// TIA Portal V18 export
ORGANIZATION_BLOCK "OLDRestart"   // OB124, LAD, ProgramCycle
TITLE = "Main Program Sweep (Cycle)"
{ S7_Optimized_Access := 'TRUE' }
VERSION : 0.1
// stored: AutoNumber true, IsIECCheckEnabled false, SetENOAutomatically false
   VAR_INPUT
      Initial_Call : Bool;   // Initial call of this OB
      Remanence : Bool;   // =True, if remanent data are available
   END_VAR
BEGIN

REGION Network 1: RESTART CMMO Z2
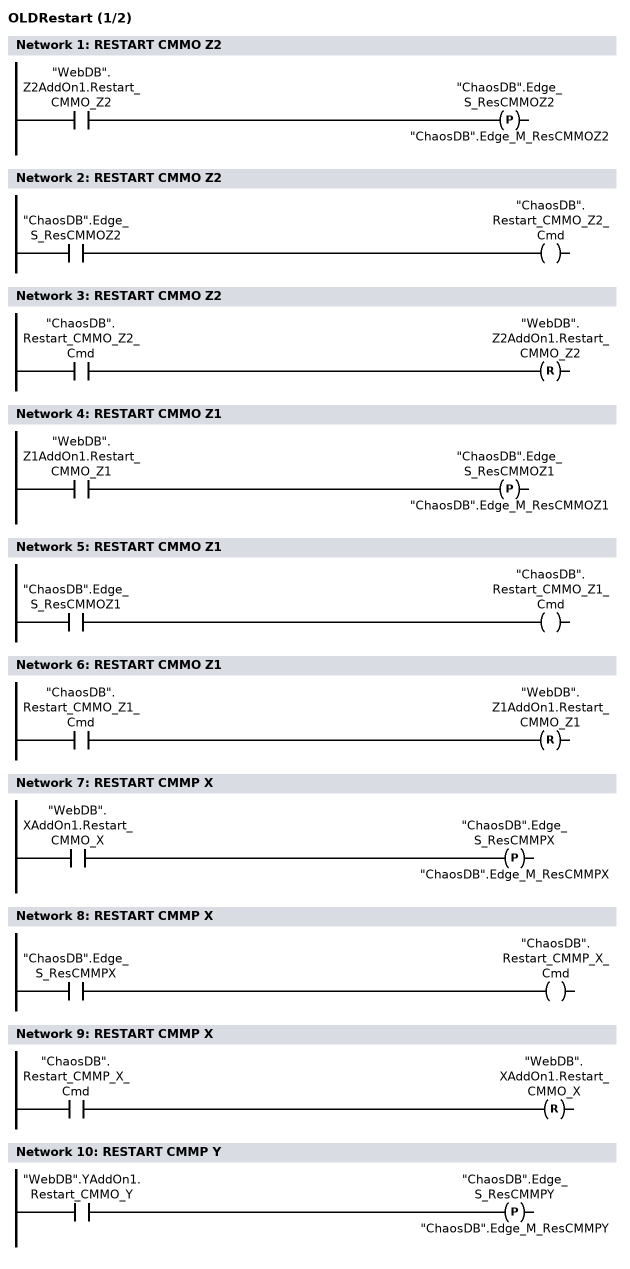
   "ChaosDB".Edge_S_ResCMMOZ2 := "WebDB".Z2AddOn1.Restart_CMMO_Z2 AND NOT "ChaosDB".Edge_M_ResCMMOZ2;   // rising edge
   "ChaosDB".Edge_M_ResCMMOZ2 := "WebDB".Z2AddOn1.Restart_CMMO_Z2;
END_REGION

REGION Network 2: RESTART CMMO Z2
   RUNG wire#powerrail
      Contact( "ChaosDB".Edge_S_ResCMMOZ2 )
      Coil( "ChaosDB".Restart_CMMO_Z2_Cmd )
   END_RUNG
   // the same network as SCL:
   "ChaosDB".Restart_CMMO_Z2_Cmd := "ChaosDB".Edge_S_ResCMMOZ2;
END_REGION

REGION Network 3: RESTART CMMO Z2
   RUNG wire#powerrail
      Contact( "ChaosDB".Restart_CMMO_Z2_Cmd )
      R_Coil( "WebDB".Z2AddOn1.Restart_CMMO_Z2 )
   END_RUNG
   // the same network as SCL:
   IF "ChaosDB".Restart_CMMO_Z2_Cmd THEN "WebDB".Z2AddOn1.Restart_CMMO_Z2 := FALSE; END_IF;
END_REGION

REGION Network 4: RESTART CMMO Z1
   "ChaosDB".Edge_S_ResCMMOZ1 := "WebDB".Z1AddOn1.Restart_CMMO_Z1 AND NOT "ChaosDB".Edge_M_ResCMMOZ1;   // rising edge
   "ChaosDB".Edge_M_ResCMMOZ1 := "WebDB".Z1AddOn1.Restart_CMMO_Z1;
END_REGION

REGION Network 5: RESTART CMMO Z1
   RUNG wire#powerrail
      Contact( "ChaosDB".Edge_S_ResCMMOZ1 )
      Coil( "ChaosDB".Restart_CMMO_Z1_Cmd )
   END_RUNG
   // the same network as SCL:
   "ChaosDB".Restart_CMMO_Z1_Cmd := "ChaosDB".Edge_S_ResCMMOZ1;
END_REGION

REGION Network 6: RESTART CMMO Z1
   RUNG wire#powerrail
      Contact( "ChaosDB".Restart_CMMO_Z1_Cmd )
      R_Coil( "WebDB".Z1AddOn1.Restart_CMMO_Z1 )
   END_RUNG
   // the same network as SCL:
   IF "ChaosDB".Restart_CMMO_Z1_Cmd THEN "WebDB".Z1AddOn1.Restart_CMMO_Z1 := FALSE; END_IF;
END_REGION

REGION Network 7: RESTART CMMP X
   "ChaosDB".Edge_S_ResCMMPX := "WebDB".XAddOn1.Restart_CMMO_X AND NOT "ChaosDB".Edge_M_ResCMMPX;   // rising edge
   "ChaosDB".Edge_M_ResCMMPX := "WebDB".XAddOn1.Restart_CMMO_X;
END_REGION

REGION Network 8: RESTART CMMP X
   RUNG wire#powerrail
      Contact( "ChaosDB".Edge_S_ResCMMPX )
      Coil( "ChaosDB".Restart_CMMP_X_Cmd )
   END_RUNG
   // the same network as SCL:
   "ChaosDB".Restart_CMMP_X_Cmd := "ChaosDB".Edge_S_ResCMMPX;
END_REGION

REGION Network 9: RESTART CMMP X
   RUNG wire#powerrail
      Contact( "ChaosDB".Restart_CMMP_X_Cmd )
      R_Coil( "WebDB".XAddOn1.Restart_CMMO_X )
   END_RUNG
   // the same network as SCL:
   IF "ChaosDB".Restart_CMMP_X_Cmd THEN "WebDB".XAddOn1.Restart_CMMO_X := FALSE; END_IF;
END_REGION

REGION Network 10: RESTART CMMP Y
   "ChaosDB".Edge_S_ResCMMPY := "WebDB".YAddOn1.Restart_CMMO_Y AND NOT "ChaosDB".Edge_M_ResCMMPY;   // rising edge
   "ChaosDB".Edge_M_ResCMMPY := "WebDB".YAddOn1.Restart_CMMO_Y;
END_REGION

REGION Network 11: RESTART CMMP Y
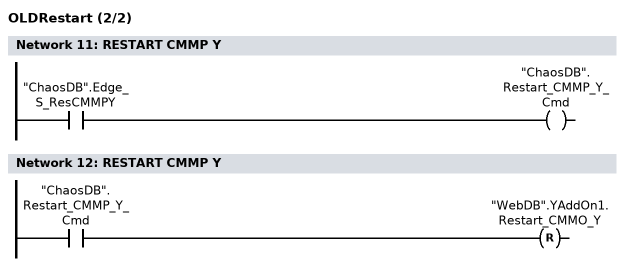
   RUNG wire#powerrail
      Contact( "ChaosDB".Edge_S_ResCMMPY )
      Coil( "ChaosDB".Restart_CMMP_Y_Cmd )
   END_RUNG
   // the same network as SCL:
   "ChaosDB".Restart_CMMP_Y_Cmd := "ChaosDB".Edge_S_ResCMMPY;
END_REGION

REGION Network 12: RESTART CMMP Y
   RUNG wire#powerrail
      Contact( "ChaosDB".Restart_CMMP_Y_Cmd )
      R_Coil( "WebDB".YAddOn1.Restart_CMMO_Y )
   END_RUNG
   // the same network as SCL:
   IF "ChaosDB".Restart_CMMP_Y_Cmd THEN "WebDB".YAddOn1.Restart_CMMO_Y := FALSE; END_IF;
END_REGION
END_ORGANIZATION_BLOCK
